// TIA Portal V15.1 export
// export: Created 2024-06-21T08:41:02.1743817Z, ExportSetting WithDefaults, DisplayName Totally Integrated Automation Portal, DisplayVersion V15.1 Update 5, DisplayName TIA Portal Openness, DisplayVersion V15.1 Update 5, DisplayName SINAMICS Startdrive Advanced, DisplayVersion V15.1, DisplayName G130, G150, S120, S150, SINAMICS MV, S210, DisplayVersion V15.1, DisplayName G110M, G120, G120C, G120D, G120P, DisplayVersion V15.1, DisplayName STEP 7 Professional, DisplayVersion V15.1 Update 5, DisplayName STEP 7 Safety, DisplayVersion V15.1, DisplayName WinCC Professional, DisplayVersion V15.1 Update 5, DisplayName SIMATIC Visualization Architect, DisplayVersion V15.1
FUNCTION_BLOCK "LProcProdMode"   // FB1716, FBD
TITLE = LProcProductionMode
{ S7_Optimized_Access := 'FALSE' }
AUTHOR : VCC
FAMILY : Control
NAME : PrProdMo
VERSION : 1.0
// ================================================================================
// This module handles all production modes for a process modezone. The production 
// modes are Weekend, Maintenance and Production Stop.
// ================================================================================
// stored: AutoNumber false, IsIECCheckEnabled false, SetENOAutomatically False, UDAEnableTagReadback false
   VAR_INPUT
      I_ExtWeekendReq { ExternalAccessible := 'False'; ExternalVisible := 'False'; ExternalWritable := 'False'} : Bool;   // External bypass request
      I_WeekendReached { ExternalAccessible := 'False'; ExternalVisible := 'False'; ExternalWritable := 'False'} : Bool;   // Weekend reached
      I_ExtMaintReq { ExternalAccessible := 'False'; ExternalVisible := 'False'; ExternalWritable := 'False'} : Bool;   // External Maintenance request
      I_MaintReached { ExternalAccessible := 'False'; ExternalVisible := 'False'; ExternalWritable := 'False'} : Bool;   // Maintenance reached
      I_ExtProdStpReq { ExternalAccessible := 'False'; ExternalVisible := 'False'; ExternalWritable := 'False'} : Bool;   // External production stop request
      I_ProdStpReached { ExternalAccessible := 'False'; ExternalVisible := 'False'; ExternalWritable := 'False'} : Bool;   // Production mode reached
   END_VAR
   VAR_OUTPUT
      O_ProcProdMode { ExternalAccessible := 'False'; ExternalVisible := 'False'; ExternalWritable := 'False'} : Word;   // Prodution Modes
      O_WeekendModeSel { ExternalAccessible := 'False'; ExternalVisible := 'False'; ExternalWritable := 'False'} : Bool;   // Weekend mode selected
      O_WeekendMode { ExternalAccessible := 'False'; ExternalVisible := 'False'; ExternalWritable := 'False'} : Bool;   // Weekend mode active
      O_MaintModeSel { ExternalAccessible := 'False'; ExternalVisible := 'False'; ExternalWritable := 'False'} : Bool;   // Maintenance mode selected
      O_MaintMode { ExternalAccessible := 'False'; ExternalVisible := 'False'; ExternalWritable := 'False'} : Bool;   // Maintenance mode active
      O_ProdStpModeSel { ExternalAccessible := 'False'; ExternalVisible := 'False'; ExternalWritable := 'False'} : Bool;   // Production mode selected
      O_ProdStpMode { ExternalAccessible := 'False'; ExternalVisible := 'False'; ExternalWritable := 'False'} : Bool;   // Production mode active
      O_AnyProdModeSel { ExternalAccessible := 'False'; ExternalVisible := 'False'; ExternalWritable := 'False'} : Bool;   // Any production mode selected
      O_AnyProdModeActive { ExternalAccessible := 'False'; ExternalVisible := 'False'; ExternalWritable := 'False'} : Bool;   // Any production mode active
      O_AlarmABCondition { ExternalAccessible := 'False'; ExternalVisible := 'False'; ExternalWritable := 'False'} : Bool;   // Alarm AB condition
      O_AlarmA { ExternalAccessible := 'False'; ExternalVisible := 'False'; ExternalWritable := 'False'} : Bool;   // Alarms A
      O_AlarmB { ExternalAccessible := 'False'; ExternalVisible := 'False'; ExternalWritable := 'False'} : Bool;   // Alarms B
      O_AlarmC { ExternalAccessible := 'False'; ExternalVisible := 'False'; ExternalWritable := 'False'} : Bool;   // Alarms C
      O_AlarmD { ExternalAccessible := 'False'; ExternalVisible := 'False'; ExternalWritable := 'False'} : Bool;   // Alarms D
      H_AlarmWord { ExternalAccessible := 'False'; ExternalVisible := 'False'; ExternalWritable := 'False'} : DWord;   // Alarm Word
   END_VAR
   VAR DB_SPECIFIC
      AD_WESelected { ExternalAccessible := 'False'; ExternalVisible := 'False'; ExternalWritable := 'False'} : Bool;   // Week-end mode selected
      AD_MaintSelected { ExternalAccessible := 'False'; ExternalVisible := 'False'; ExternalWritable := 'False'} : Bool;   // Maintenance mode selected
      AD_ProdStopSelected { ExternalAccessible := 'False'; ExternalVisible := 'False'; ExternalWritable := 'False'} : Bool;   // Production mode selected
      H_HMIProcModeCmd : Word;   // Production mode commands from HMI
      H_Anim : Word;   // Animation
      HMIWeekendReq { ExternalAccessible := 'False'; ExternalVisible := 'False'; ExternalWritable := 'False'} : Bool;   // Bypass selected on HMI
      HMIMaintReq { ExternalAccessible := 'False'; ExternalVisible := 'False'; ExternalWritable := 'False'} : Bool;   // Maintenance selected on HMI
      HMIProdStpReq { ExternalAccessible := 'False'; ExternalVisible := 'False'; ExternalWritable := 'False'} : Bool;   // Production mode selected on HMI
      WeekendSelected { ExternalAccessible := 'False'; ExternalVisible := 'False'; ExternalWritable := 'False'} : Bool;   // Weekend is selected
      MaintSelected { ExternalAccessible := 'False'; ExternalVisible := 'False'; ExternalWritable := 'False'} : Bool;   // Maintenance is selected
      ProdStpSelected { ExternalAccessible := 'False'; ExternalVisible := 'False'; ExternalWritable := 'False'} : Bool;   // Production stop is selected
      WeekendActive { ExternalAccessible := 'False'; ExternalVisible := 'False'; ExternalWritable := 'False'} : Bool;   // Weekend is active
      MaintActive { ExternalAccessible := 'False'; ExternalVisible := 'False'; ExternalWritable := 'False'} : Bool;   // Maintenance is active
      ProdStpActive { ExternalAccessible := 'False'; ExternalVisible := 'False'; ExternalWritable := 'False'} : Bool;   // Production stop is active
      TmpMaintReqOff { ExternalAccessible := 'False'; ExternalVisible := 'False'; ExternalWritable := 'False'} : Bool;   // Temporary request off
      TmpMaintReqOn { ExternalAccessible := 'False'; ExternalVisible := 'False'; ExternalWritable := 'False'} : Bool;   // Temporary request on
      PulseMaintReqOn { ExternalAccessible := 'False'; ExternalVisible := 'False'; ExternalWritable := 'False'} : Bool;   // Pulse request on
      PulseMaintReqOff { ExternalAccessible := 'False'; ExternalVisible := 'False'; ExternalWritable := 'False'} : Bool;   // Pulse request off
      TmpWeekendReqOff { ExternalAccessible := 'False'; ExternalVisible := 'False'; ExternalWritable := 'False'} : Bool;   // Temporary request off
      TmpWeekendReqOn { ExternalAccessible := 'False'; ExternalVisible := 'False'; ExternalWritable := 'False'} : Bool;   // Temporary request on
      PulseWeekendReqOn { ExternalAccessible := 'False'; ExternalVisible := 'False'; ExternalWritable := 'False'} : Bool;   // Pulse request on
      PulseWeekendReqOff { ExternalAccessible := 'False'; ExternalVisible := 'False'; ExternalWritable := 'False'} : Bool;   // Pulse request off
      TmpProdStpReqOff { ExternalAccessible := 'False'; ExternalVisible := 'False'; ExternalWritable := 'False'} : Bool;   // Temporary request off
      TmpProdStpReqOn { ExternalAccessible := 'False'; ExternalVisible := 'False'; ExternalWritable := 'False'} : Bool;   // Temporary request on
      PulseProdStpReqOn { ExternalAccessible := 'False'; ExternalVisible := 'False'; ExternalWritable := 'False'} : Bool;   // Pulse request on
      PulseProdStpReqOff { ExternalAccessible := 'False'; ExternalVisible := 'False'; ExternalWritable := 'False'} : Bool;   // Pulse request off
      AlarmA { ExternalAccessible := 'False'; ExternalVisible := 'False'; ExternalWritable := 'False'} : Bool;   // Alarm A active in the FB
      AlarmB { ExternalAccessible := 'False'; ExternalVisible := 'False'; ExternalWritable := 'False'} : Bool;   // Alarm B active in the FB
      AlarmC { ExternalAccessible := 'False'; ExternalVisible := 'False'; ExternalWritable := 'False'} : Bool;   // Alarm C active in the FB
      AlarmD { ExternalAccessible := 'False'; ExternalVisible := 'False'; ExternalWritable := 'False'} : Bool;   // Alarm D active in the FB
   END_VAR
   VAR_TEMP   // added for the SCL form of the ladder/FBD networks
      _w1 : Bool;
      _w2 : Bool;
   END_VAR
BEGIN

REGION Network 1: **** 1 - Inputs **** Extract the production modes from HMI
   // Extract the production modes from HMI
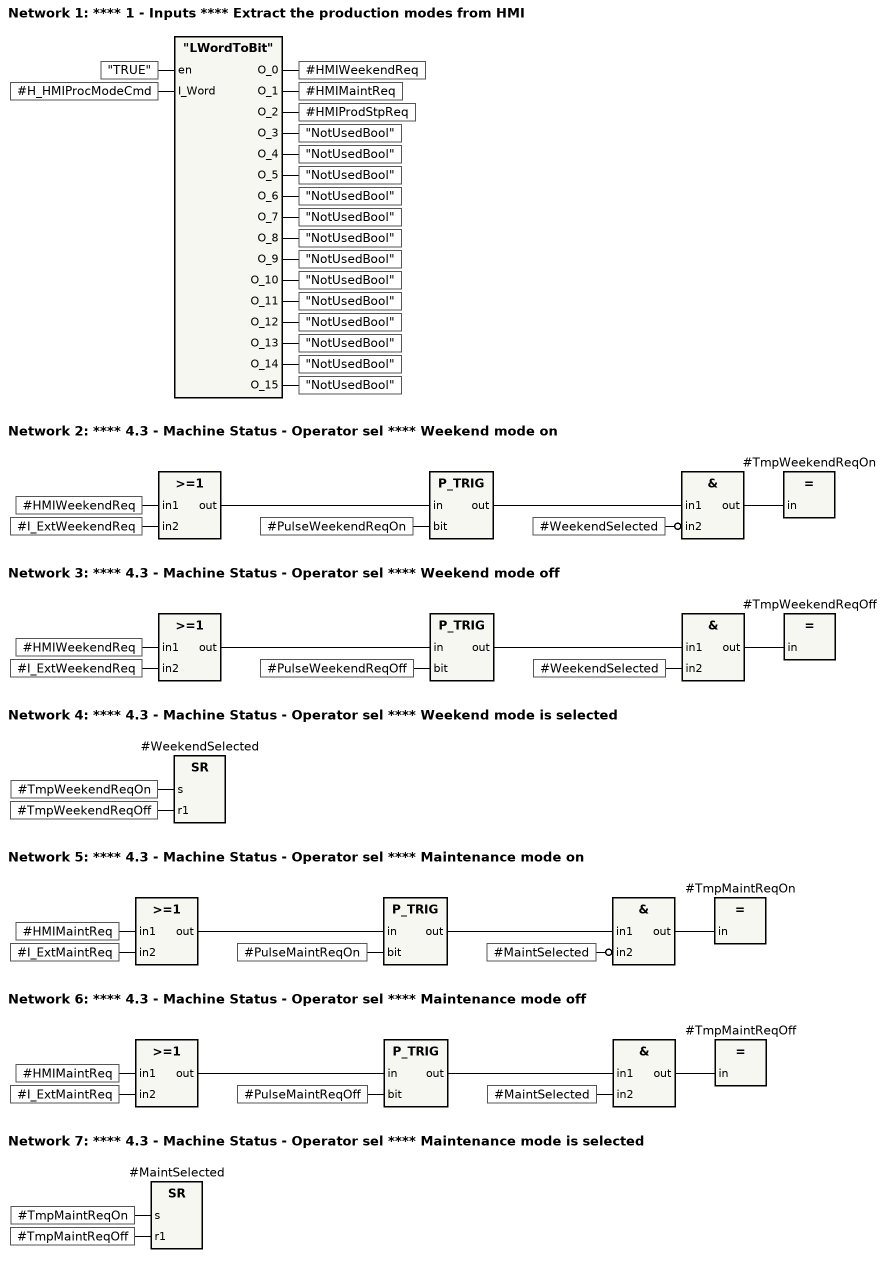
   IF "TRUE" THEN
       "LWordToBit"(I_Word := #H_HMIProcModeCmd,
                    O_0 => #HMIWeekendReq,
                    O_1 => #HMIMaintReq,
                    O_2 => #HMIProdStpReq,
                    O_3 => "NotUsedBool",
                    O_4 => "NotUsedBool",
                    O_5 => "NotUsedBool",
                    O_6 => "NotUsedBool",
                    O_7 => "NotUsedBool",
                    O_8 => "NotUsedBool",
                    O_9 => "NotUsedBool",
                    O_10 => "NotUsedBool",
                    O_11 => "NotUsedBool",
                    O_12 => "NotUsedBool",
                    O_13 => "NotUsedBool",
                    O_14 => "NotUsedBool",
                    O_15 => "NotUsedBool");
   END_IF;
END_REGION

REGION Network 2: **** 4.3 - Machine Status - Operator sel **** Weekend mode on
   // Weekend mode on
   #_w1 := #HMIWeekendReq OR #I_ExtWeekendReq;
   #_w2 := #_w1 AND NOT #PulseWeekendReqOn;   // rising edge
   #PulseWeekendReqOn := #_w1;
   #TmpWeekendReqOn := #_w2 AND NOT #WeekendSelected;
END_REGION

REGION Network 3: **** 4.3 - Machine Status - Operator sel **** Weekend mode off
   // Weekend mode off
   #_w1 := #HMIWeekendReq OR #I_ExtWeekendReq;
   #_w2 := #_w1 AND NOT #PulseWeekendReqOff;   // rising edge
   #PulseWeekendReqOff := #_w1;
   #TmpWeekendReqOff := #_w2 AND #WeekendSelected;
END_REGION

REGION Network 4: **** 4.3 - Machine Status - Operator sel **** Weekend mode is selected
   // Weekend mode is selected
   IF #TmpWeekendReqOn THEN
       #WeekendSelected := TRUE;   // SR flip-flop
   END_IF;
   IF #TmpWeekendReqOff THEN #WeekendSelected := FALSE; END_IF;
END_REGION

REGION Network 5: **** 4.3 - Machine Status - Operator sel **** Maintenance mode on
   // Maintenance mode on
   #_w1 := #HMIMaintReq OR #I_ExtMaintReq;
   #_w2 := #_w1 AND NOT #PulseMaintReqOn;   // rising edge
   #PulseMaintReqOn := #_w1;
   #TmpMaintReqOn := #_w2 AND NOT #MaintSelected;
END_REGION

REGION Network 6: **** 4.3 - Machine Status - Operator sel **** Maintenance mode off
   // Maintenance mode off
   #_w1 := #HMIMaintReq OR #I_ExtMaintReq;
   #_w2 := #_w1 AND NOT #PulseMaintReqOff;   // rising edge
   #PulseMaintReqOff := #_w1;
   #TmpMaintReqOff := #_w2 AND #MaintSelected;
END_REGION

REGION Network 7: **** 4.3 - Machine Status - Operator sel **** Maintenance mode is selected
   // Maintenance mode is selected
   IF #TmpMaintReqOn THEN
       #MaintSelected := TRUE;   // SR flip-flop
   END_IF;
   IF #TmpMaintReqOff THEN #MaintSelected := FALSE; END_IF;
END_REGION

REGION Network 8: **** 4.3 - Machine Status - Operator sel **** Production stop mode on
   // Production stop mode on
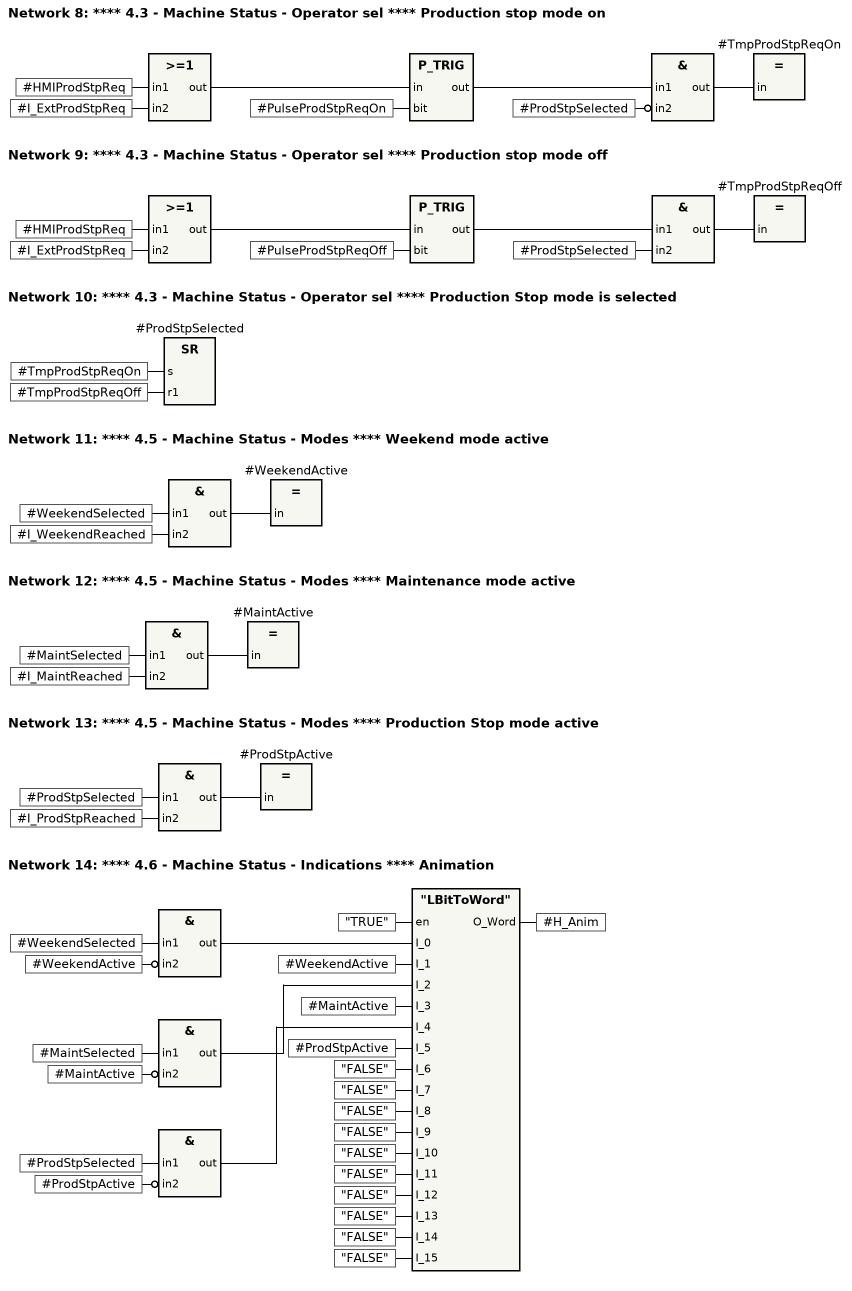
   #_w1 := #HMIProdStpReq OR #I_ExtProdStpReq;
   #_w2 := #_w1 AND NOT #PulseProdStpReqOn;   // rising edge
   #PulseProdStpReqOn := #_w1;
   #TmpProdStpReqOn := #_w2 AND NOT #ProdStpSelected;
END_REGION

REGION Network 9: **** 4.3 - Machine Status - Operator sel **** Production stop mode off
   // Production stop mode off
   #_w1 := #HMIProdStpReq OR #I_ExtProdStpReq;
   #_w2 := #_w1 AND NOT #PulseProdStpReqOff;   // rising edge
   #PulseProdStpReqOff := #_w1;
   #TmpProdStpReqOff := #_w2 AND #ProdStpSelected;
END_REGION

REGION Network 10: **** 4.3 - Machine Status - Operator sel **** Production Stop mode is selected
   // Production Stop mode is selected
   IF #TmpProdStpReqOn THEN
       #ProdStpSelected := TRUE;   // SR flip-flop
   END_IF;
   IF #TmpProdStpReqOff THEN #ProdStpSelected := FALSE; END_IF;
END_REGION

REGION Network 11: **** 4.5 - Machine Status - Modes **** Weekend mode active
   // Weekend mode active
   #WeekendActive := #WeekendSelected AND #I_WeekendReached;
END_REGION

REGION Network 12: **** 4.5 - Machine Status - Modes **** Maintenance mode active
   // Maintenance mode active
   #MaintActive := #MaintSelected AND #I_MaintReached;
END_REGION

REGION Network 13: **** 4.5 - Machine Status - Modes **** Production Stop mode active
   // Production Stop mode active
   #ProdStpActive := #ProdStpSelected AND #I_ProdStpReached;
END_REGION

REGION Network 14: **** 4.6 - Machine Status - Indications **** Animation
   // Animation
   IF "TRUE" THEN
       "LBitToWord"(I_0 := #WeekendSelected AND NOT #WeekendActive,
                    I_1 := #WeekendActive,
                    I_2 := #MaintSelected AND NOT #MaintActive,
                    I_3 := #MaintActive,
                    I_4 := #ProdStpSelected AND NOT #ProdStpActive,
                    I_5 := #ProdStpActive,
                    I_6 := "FALSE",
                    I_7 := "FALSE",
                    I_8 := "FALSE",
                    I_9 := "FALSE",
                    I_10 := "FALSE",
                    I_11 := "FALSE",
                    I_12 := "FALSE",
                    I_13 := "FALSE",
                    I_14 := "FALSE",
                    I_15 := "FALSE",
                    O_Word => #H_Anim);
   END_IF;
END_REGION

REGION Network 15: **** 8 - Outputs **** Set the different bits in the Production Mode register
   // Set the different bits in the Production Mode register
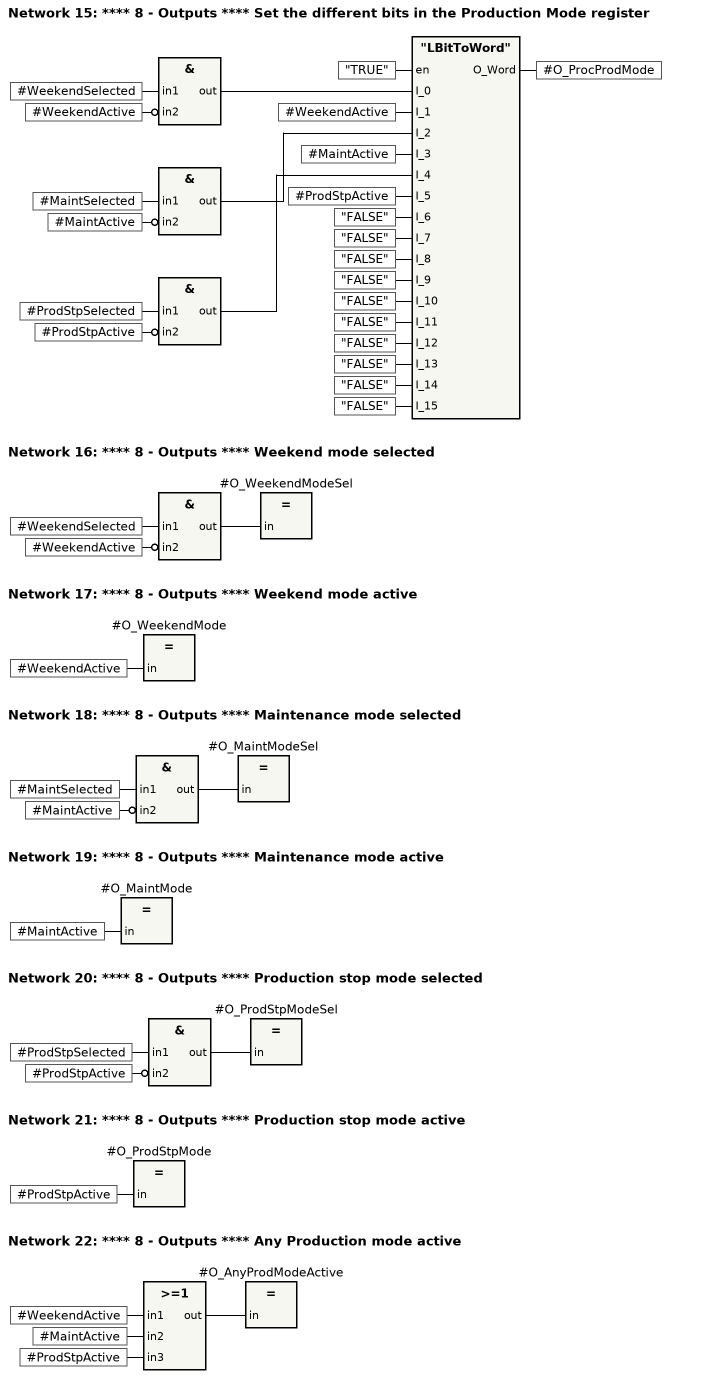
   IF "TRUE" THEN
       "LBitToWord"(I_0 := #WeekendSelected AND NOT #WeekendActive,
                    I_1 := #WeekendActive,
                    I_2 := #MaintSelected AND NOT #MaintActive,
                    I_3 := #MaintActive,
                    I_4 := #ProdStpSelected AND NOT #ProdStpActive,
                    I_5 := #ProdStpActive,
                    I_6 := "FALSE",
                    I_7 := "FALSE",
                    I_8 := "FALSE",
                    I_9 := "FALSE",
                    I_10 := "FALSE",
                    I_11 := "FALSE",
                    I_12 := "FALSE",
                    I_13 := "FALSE",
                    I_14 := "FALSE",
                    I_15 := "FALSE",
                    O_Word => #O_ProcProdMode);
   END_IF;
END_REGION

REGION Network 16: **** 8 - Outputs **** Weekend mode selected
   // Weekend mode selected
   #O_WeekendModeSel := #WeekendSelected AND NOT #WeekendActive;
END_REGION

REGION Network 17: **** 8 - Outputs **** Weekend mode active
   // Weekend mode active
   #O_WeekendMode := #WeekendActive;
END_REGION

REGION Network 18: **** 8 - Outputs **** Maintenance mode selected
   // Maintenance mode selected
   #O_MaintModeSel := #MaintSelected AND NOT #MaintActive;
END_REGION

REGION Network 19: **** 8 - Outputs **** Maintenance mode active
   // Maintenance mode active
   #O_MaintMode := #MaintActive;
END_REGION

REGION Network 20: **** 8 - Outputs **** Production stop mode selected
   // Production stop mode selected
   #O_ProdStpModeSel := #ProdStpSelected AND NOT #ProdStpActive;
END_REGION

REGION Network 21: **** 8 - Outputs **** Production stop mode active
   // Production stop mode active
   #O_ProdStpMode := #ProdStpActive;
END_REGION

REGION Network 22: **** 8 - Outputs **** Any Production mode active
   // Any Production mode active
   #O_AnyProdModeActive := #WeekendActive OR #MaintActive OR #ProdStpActive;
END_REGION

REGION Network 23: **** 8 - Outputs **** Any Production mode active
   // Any Production mode active
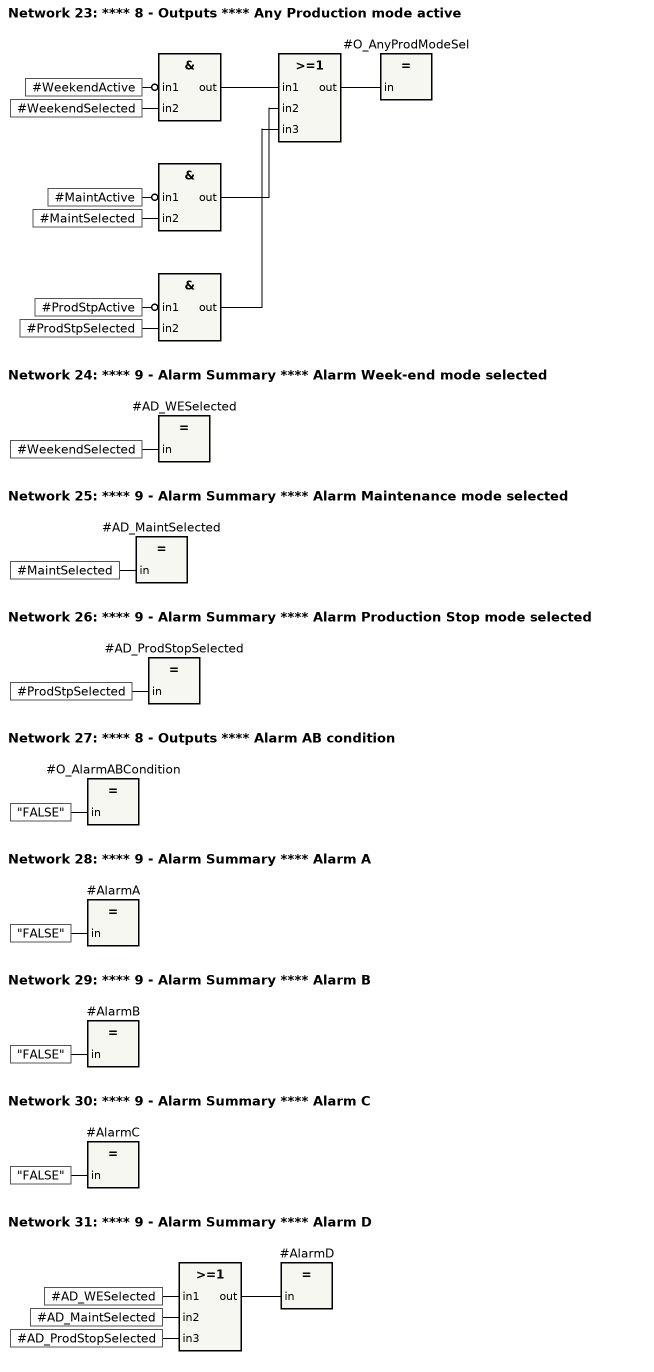
   #O_AnyProdModeSel := (NOT #WeekendActive AND #WeekendSelected) OR (NOT #MaintActive AND #MaintSelected) OR (NOT #ProdStpActive AND #ProdStpSelected);
END_REGION

REGION Network 24: **** 9 - Alarm Summary **** Alarm Week-end mode selected
   // Alarm Week-end mode selected
   #AD_WESelected := #WeekendSelected;
END_REGION

REGION Network 25: **** 9 - Alarm Summary **** Alarm Maintenance mode selected
   // Alarm Maintenance mode selected
   #AD_MaintSelected := #MaintSelected;
END_REGION

REGION Network 26: **** 9 - Alarm Summary **** Alarm Production Stop mode selected
   // Alarm Production Stop mode selected
   #AD_ProdStopSelected := #ProdStpSelected;
END_REGION

REGION Network 27: **** 8 - Outputs **** Alarm AB condition
   // Alarm AB condition
   #O_AlarmABCondition := "FALSE";
END_REGION

REGION Network 28: **** 9 - Alarm Summary **** Alarm A
   // Summary of alarms A
   #AlarmA := "FALSE";
END_REGION

REGION Network 29: **** 9 - Alarm Summary **** Alarm B
   // Summary of alarms B
   #AlarmB := "FALSE";
END_REGION

REGION Network 30: **** 9 - Alarm Summary **** Alarm C
   // Summary of alarms C
   #AlarmC := "FALSE";
END_REGION

REGION Network 31: **** 9 - Alarm Summary **** Alarm D
   // Summary of alarms D
   #AlarmD := #AD_WESelected OR #AD_MaintSelected OR #AD_ProdStopSelected;
END_REGION

REGION Network 32: **** 9.1 - Alarm Output **** Alarm A
   // Summary of alarms A
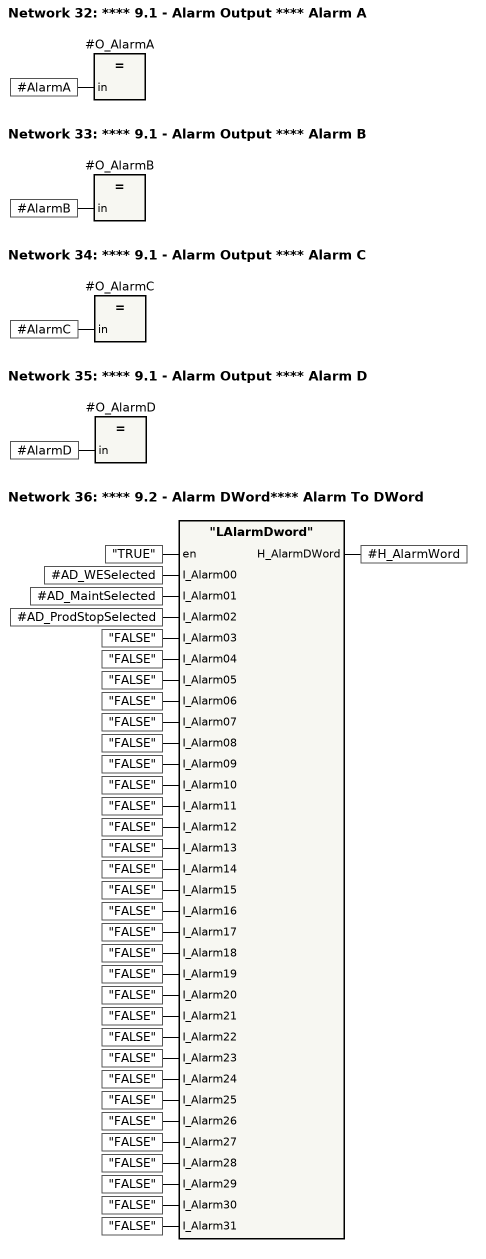
   #O_AlarmA := #AlarmA;
END_REGION

REGION Network 33: **** 9.1 - Alarm Output **** Alarm B
   // Summary of alarms B
   #O_AlarmB := #AlarmB;
END_REGION

REGION Network 34: **** 9.1 - Alarm Output **** Alarm C
   // Summary of alarms C
   #O_AlarmC := #AlarmC;
END_REGION

REGION Network 35: **** 9.1 - Alarm Output **** Alarm D
   // Summary of alarms D
   #O_AlarmD := #AlarmD;
END_REGION

REGION Network 36: **** 9.2 - Alarm DWord**** Alarm To DWord
   // Alarm Word
   IF "TRUE" THEN
       "LAlarmDword"(I_Alarm00 := #AD_WESelected,
                     I_Alarm01 := #AD_MaintSelected,
                     I_Alarm02 := #AD_ProdStopSelected,
                     I_Alarm03 := "FALSE",
                     I_Alarm04 := "FALSE",
                     I_Alarm05 := "FALSE",
                     I_Alarm06 := "FALSE",
                     I_Alarm07 := "FALSE",
                     I_Alarm08 := "FALSE",
                     I_Alarm09 := "FALSE",
                     I_Alarm10 := "FALSE",
                     I_Alarm11 := "FALSE",
                     I_Alarm12 := "FALSE",
                     I_Alarm13 := "FALSE",
                     I_Alarm14 := "FALSE",
                     I_Alarm15 := "FALSE",
                     I_Alarm16 := "FALSE",
                     I_Alarm17 := "FALSE",
                     I_Alarm18 := "FALSE",
                     I_Alarm19 := "FALSE",
                     I_Alarm20 := "FALSE",
                     I_Alarm21 := "FALSE",
                     I_Alarm22 := "FALSE",
                     I_Alarm23 := "FALSE",
                     I_Alarm24 := "FALSE",
                     I_Alarm25 := "FALSE",
                     I_Alarm26 := "FALSE",
                     I_Alarm27 := "FALSE",
                     I_Alarm28 := "FALSE",
                     I_Alarm29 := "FALSE",
                     I_Alarm30 := "FALSE",
                     I_Alarm31 := "FALSE",
                     H_AlarmDWord => #H_AlarmWord);
   END_IF;
END_REGION
END_FUNCTION_BLOCK
